Yaskawa INFORM job: TESTR.JBI

/JOB
//NAME TESTR
//POS
///NPOS 1,1,0,0,0,0
///TOOL 0
///POSTYPE BASE
///RECTAN
///RCONF 0,0,0,0,0,0,0,0,0,0,0,0,0,0,0,0,0,0,0,0,0,0,0,0
C00000=1790.554,5112.321,-676.984,1.1183,49.7665,-139.7613
BC00000=1011.689,4837.660,450.143
//INST
///DATE 2024/01/25 09:47
///ATTR SC,RW,RJ
////FRAME BASE
///GROUP1 RB1,BS1
NOP
MOVJ C00000 BC00000 VJ=0.78
END
